SUBAPPLICATION logiBUS_AI_Raw_VT_AR_OPC (* logiBUS_AI_IDA (Analog-Eingang, lokal) lesen -> Rohwert per OPC-UA publizieren (REAL 0-4095) + VT-Zahlenfeld (Rohwert, reine Diagnose-Anzeige) -> als AR-Plug ausgeben, fertig zur Weiterverarbeitung durch einen Kalibrier-Baustein (AR_CALIBRATE_2P_REF.X / AR_CALIBRATE_3P_REF.X). Herausgeloest aus logiBUS_AI_Calibrate_IDA_OPC/_3P_IDA_OPC (logiBUS_AI_IDA+AD_TO_AUDI+AUDI_SPLIT_2+Q_NumericValue_RAW+AUDI_TO_AR kam dort 2x identisch vor). *)
  (* Standard: 61499-2; Description: Copyright (c) 2026 Meisterschulen am Ostbahnhof This program and the accompanying materials are made available under the terms of the Eclipse Public License 2.0 which is available at https://www.eclipse.org/legal/epl-2.0/ SPDX-License-Identifier: EPL-2.0 *)
  (* Version 1.1, 2026-09-27, Franz Höpfinger, Meisterschulen am Ostbahnhof, Bugfix (Live-Log STG1): 'RD_0 of FB ...RawDisplay.AR_SUBSCRIBE_M2M.SUBSCRIBE_1 has no data, is not a scalar or there is a type mismatch', 170x im Log, auf allen 5 co-located Sensor-Stationen (Fuellband/Schnitthoehe/Druck/Oeltemperatur/Hangausgleich Winkel). Ursache: ID_RAW_WRITE ging bisher per AD_PUBLISH_1 (DWORD) raus, aber die STG1-Seite (AR_M2M_Subscribe_TO_Q_Publish_OPC.RawDisplay) abonniert per AR_SUBSCRIBE_1 (REAL) - Typkonflikt auf dem Draht. Zero-Raw/Span-Raw (an den Kalibrierpunkten) hatten dasselbe Problem nie, weil die schon immer per AR_PUBLISH_1 (REAL) rausgehen. AD_SPLIT_2/AD_PUBLISH_RAW entfernt, AR_OUT jetzt per neuem AR_SPLIT_2_Raw zusaetzlich an neuen AR_PUBLISH_RAW (AR_PUBLISH_1) verzweigt - ACHTUNG: aendert den OPC-UA-Datentyp auf dem Draht, alle Stationen mit einer Calibrate_2P/3P_IDA_OPC-Instanz (STG2/STG3/STG4) muessen neu gebaut UND geflasht werden, nicht nur STG1. *)
  (* Version 1.0, 2026-09-18, Franz Höpfinger, Meisterschulen am Ostbahnhof, initial implementation - herausgeloest aus logiBUS_AI_Calibrate_IDA_OPC/_3P_IDA_OPC, wiederverwendbar fuer jeden lokal (auf derselben Station wie die VT) angeschlossenen Analog-Eingang mit Rohwert-Publish+VT-Anzeige, unabhaengig von 2- oder 3-Punkt-Kalibrierung. *)
  PACKAGE MyLib::sys;
  IMPORT logiBUS::io::AI::logiBUS_AI;
  IMPORT logiBUS::io::AI::logiBUS_AI_S;
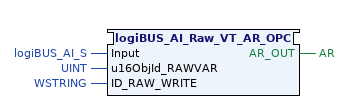
  VAR_INPUT
    Input : logiBUS::io::AI::logiBUS_AI_S := logiBUS_AI::Invalid; (* Identify the Input AnalogInput_I1..I8 *)
    u16ObjId_RAWVAR : UINT; (* Object ID CNumberVariable (Rohwert 0-4095, unkalibriert, reine Diagnose-Anzeige) *)
    ID_RAW_WRITE : WSTRING; (* Rohwert-Ruckmelde-Adresse (REAL 0-4095, ACTION=PUBLISH) *)
  END_VAR
  PLUGS
    AR_OUT : adapter::types::unidirectional::AR; (* Rohwert als AR, fertig fuer CALIBRATE.X *)
  END_PLUGS
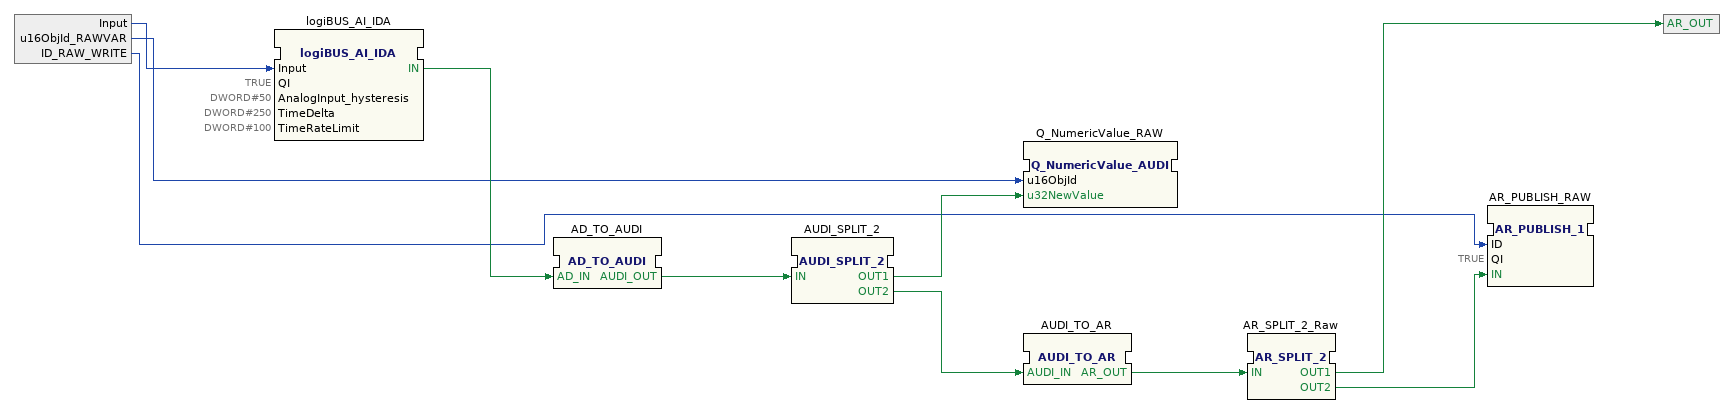
  FBS
    logiBUS_AI_IDA : logiBUS::io::AI::logiBUS_AI_IDA(QI := TRUE, AnalogInput_hysteresis := DWORD#50, TimeDelta := DWORD#250, TimeRateLimit := DWORD#100);
    AD_TO_AUDI : adapter::conversion::unidirectional::AD_TO_AUDI;
    AUDI_SPLIT_2 : adapter::events::unidirectional::AUDI_SPLIT_2;
    Q_NumericValue_RAW : isobus::UT::Q::Q_NumericValue_AUDI;
    AUDI_TO_AR : adapter::conversion::unidirectional::AUDI_TO_AR;
    AR_SPLIT_2_Raw : adapter::events::unidirectional::AR_SPLIT_2;
    AR_PUBLISH_RAW : adapter::net::AR_PUBLISH_1(QI := TRUE);
  END_FBS
  DATA_CONNECTIONS
    Input TO logiBUS_AI_IDA.Input;
    u16ObjId_RAWVAR TO Q_NumericValue_RAW.u16ObjId;
    ID_RAW_WRITE TO AR_PUBLISH_RAW.ID;
  END_CONNECTIONS
  ADAPTER_CONNECTIONS
    logiBUS_AI_IDA.IN TO AD_TO_AUDI.AD_IN;
    AD_TO_AUDI.AUDI_OUT TO AUDI_SPLIT_2.IN;
    AUDI_SPLIT_2.OUT1 TO Q_NumericValue_RAW.u32NewValue;
    AUDI_SPLIT_2.OUT2 TO AUDI_TO_AR.AUDI_IN;
    AUDI_TO_AR.AR_OUT TO AR_SPLIT_2_Raw.IN;
    AR_SPLIT_2_Raw.OUT1 TO AR_OUT;
    AR_SPLIT_2_Raw.OUT2 TO AR_PUBLISH_RAW.IN;
  END_CONNECTIONS
END_SUBAPPLICATION
